FUNCTION_BLOCK TransferToLeftorRight
VAR_INPUT
END_VAR
VAR_OUTPUT
END_VAR
VAR
	LeftExitPosEdge: R_TRIG;
	LeftExitPositive: BOOL;
	RightExitPosEdge: R_TRIG;
	RightExitPositive: BOOL;
	LeftConveyorCounter: CTUD;
	RightConveyorCounter: CTUD;
	BoxCounter: CTU;
END_VAR


//Positive edges of the sensors.
LeftExitPosEdge(CLK:= At_Left_Exit, Q=> LeftExitPositive );
RightExitPosEdge(CLK:= At_Right_Exit, Q=> RightExitPositive);
//Left conveyor box counter.
LeftConveyorCounter(
	CU:= NOT At_Left_Entry , 
	CD:= LeftExitPositive, 
	RESET:= EmergencyActivated, 
	LOAD:= , 
	PV:= , 
	QU=> , 
	QD=> , 
	CV=> );
//Right conveyor box counter.	
RightConveyorCounter(
	CU:= NOT At_Right_Entry, 
	CD:= RightExitPositive, 
	RESET:= EmergencyActivated, 
	LOAD:= , 
	PV:= , 
	QU=> , 
	QD=> , 
	CV=> );
//Left conveyor works until it is empty.
IF NOT LeftConveyorCounter.QD THEN
	Conveyor_Left := TRUE;
ELSE
	Conveyor_Left := FALSE;
END_IF
//Right conveyor works until it is empty.
IF NOT RightConveyorCounter.QD THEN
	Conveyor_Right := TRUE;
ELSE
	Conveyor_Right := FALSE;
END_IF
//Total box counter.
BoxCounter(
	CU:= LeftExitPositive OR RightExitPositive, 
	RESET:= EmergencyActivated, 
	PV:= , 
	Q=> , 
	CV=> );

BoxCounted := BoxCounter.CV;

END_FUNCTION_BLOCK

(* stored: Version 1.1.0.1, ProductVersion 3.1.4024.6
   POU TransferToLeftorRight: Id {174d7582-74a9-42e6-9100-ae2e28b59a99}, SpecialFunc None *)
